{attribute 'obsolete' := 'Use FB_PositionStatePMPS1D instead'}
FUNCTION_BLOCK FB_PositionStateBase_WithPMPS EXTENDS FB_PositionStateBase
(*
    Handles EPICS moves between multiple states for a single axis with PMPS.
    Should be subclassed for a specific enumSet and enumGet.
    See body comment  or FB_PositionStateInOut_WithPMPS for an implementation example.
*)
VAR_IN_OUT
    fbArbiter: FB_Arbiter;
    fbFFHWO: FB_HardwareFFOutput;
END_VAR
VAR_INPUT
    sPmpsDeviceName: STRING;
    sTransitionKey: STRING;
    {attribute 'pytmc' := '
        pv: PMPS:ARB:ENABLE
        io: io
    '}
    bArbiterEnabled: BOOL := TRUE;
    tArbiterTimeout: TIME := T#1s;
    bMoveOnArbiterTimeout: BOOL := TRUE;
    fStateBoundaryDeadband: LREAL := 0;
    bBPOKAutoReset: BOOL := False;
END_VAR
VAR
    {attribute 'pytmc' := 'pv: PMPS'}
    fbStatePMPS: FB_PositionStatePMPS;
    fbEncErrFFO: FB_EncErrorFFO;
END_VAR


(*
    Subclass me, define enums to translate setState and getState, call Exec

    Example:

    <something to fill arrStates>
    setState := enumSet;
    Exec();
    enumGet := getState;
    enumSet := setState;
*)

ACTION Exec:

StateHandler();
PMPSHandler();
END_ACTION

ACTION PMPSHandler:

fbStatePMPS(
    fbArbiter:=fbArbiter,
    fbFFHWO:=fbFFHWO,
    stMotionStage:=stMotionStage,
    arrStates:=arrStates,
    sPmpsDeviceName:=sPmpsDeviceName,
    sTransitionKey:=sTransitionKey,
    stPmpsDoc:= PMPS_GVL.BP_jsonDoc,
    bRequestTransition:=setState <> 0,
    setState:=setState,
    getState:=getState,
    bArbiterEnabled:=bArbiterEnabled,
    tArbiterTimeout:=tArbiterTimeout,
    bMoveOnArbiterTimeout:=bMoveOnArbiterTimeout,
    fStateBoundaryDeadband:=fStateBoundaryDeadband,
    bBPOKAutoReset:=bBPOKAutoReset);

fbEncErrFFO(
    stMotionStage:=stMotionStage,
    fbFFHWO:=fbFFHWO,
    bAutoReset:=TRUE);
END_ACTION

END_FUNCTION_BLOCK

(* stored: Version 1.1.0.1
   POU FB_PositionStateBase_WithPMPS: Id {b19911a0-9c0b-43b8-8cb3-dd3526519e98}, SpecialFunc None
   Action Exec: Id {70fa5ddc-d7df-4f92-a75a-307938fa5e37}
   Action PMPSHandler: Id {71f52474-b96e-45d5-8d7a-c1880d7070ba} *)
